// TwinCAT 3 PLC project EncapsulationPractice
// ProgramVersion: 3.1.4024.0
// libraries:
//   Tc2_Standard, * (Beckhoff Automation GmbH)
//   Tc2_System, * (Beckhoff Automation GmbH)
//   Tc3_Module, * (Beckhoff Automation GmbH)
// project tree:
//   / PlcTask.TcTTO
//   POUs/ Condition.TcPOU, FB_Bank.TcPOU, FB_IciciBank.TcPOU, MAIN.TcPOU
// (motion and I/O tree: see PLC project functionblockpractice)
// real-time tasks:
//   TASK PlcTask: cycle T#10ms, priority 20, ADS port 350
//   TASK PlcTask2: cycle T#10ms, priority 22, ADS port 352
//   TASK PlcTask1: cycle T#10ms, priority 21, ADS port 351
//   TASK PlcTask3: cycle T#10ms, priority 23, ADS port 353
//   TASK PlcTask4: cycle T#10ms, priority 24, ADS port 354
//   TASK PlcTask5: cycle T#10ms, priority 25, ADS port 355
//   TASK PlcTask6: cycle T#10ms, priority 26, ADS port 356

CONFIGURATION EncapsulationPractice
    RESOURCE PLC ON TwinCAT3
        TASK PlcTask(INTERVAL := T#10ms, PRIORITY := 25);
        PROGRAM MAIN WITH PlcTask : MAIN;
        PROGRAM Condition WITH PlcTask : Condition;
    END_RESOURCE
END_CONFIGURATION

// ---- POUs/MAIN.TcPOU
PROGRAM MAIN
VAR
	fAmount1 : REAL;
	fAmount2 : REAL;
	fbBank : FB_Bank;
	fbIciciBank : FB_IciciBank;
END_VAR

fAmount1 := fbBank.fMoney;
fbBank.sBankName := 'sbi';
fbBank.M_Deposit(4000);
fbBank.M_Withdrawal(2000);

fAmount2 := fbIciciBank.fMoney;
fbIciciBank.sBankName := 'icici';
fbIciciBank.M_Deposit(4000);
fbIciciBank.M_Withdrawal(2000);

END_PROGRAM

// ---- POUs/FB_Bank.TcPOU
FUNCTION_BLOCK FB_Bank
VAR_INPUT
	sBankName : STRING(200);
END_VAR

VAR
	fBalance : REAL;
END_VAR

{attribute 'monitoring' := 'call'}
PROPERTY fMoney : REAL
GET
fMoney := fBalance;
END_GET
SET // PRIVATE
fBalance := fMoney;
END_SET
END_PROPERTY

METHOD M_Deposit : BOOL
VAR_INPUT
	fDepositAmount : REAL;
END_VAR
fMoney := fDepositAmount;
END_METHOD

METHOD M_Withdrawal : BOOL
VAR_INPUT
	fWithdrawAmount : REAL;
END_VAR
IF fWithdrawAmount <= fMoney THEN
	fMoney := fMoney - fWithdrawAmount;
END_IF
END_METHOD

END_FUNCTION_BLOCK

// ---- POUs/FB_IciciBank.TcPOU
FUNCTION_BLOCK FB_IciciBank EXTENDS FB_Bank

VAR
END_VAR

METHOD FINAL M_Deposit : BOOL
VAR_INPUT
	fDepositAmount : REAL;
END_VAR
END_METHOD

END_FUNCTION_BLOCK

// ---- POUs/Condition.TcPOU
PROGRAM Condition
VAR
	nMark : INT := 88;
	sGrade : STRING ;
END_VAR

ACT_Case();

ACTION ACT_Case:
CASE nMark OF
	 91..100:
	sGrade := 'A';
	81..90 :
	sGrade:= 'B';
	71..80:
	sGrade:= 'C';
	61..70:
	sGrade:= 'D';
	ELSE
		sGrade:= 'F';
	
END_CASE
END_ACTION

ACTION ACT_Condition:
IF nMark > 90 THEN
	sGrade := 'A';
	ELSIF nMark > 80 THEN
		IF nMark > 85 THEN
			sGrade := 'B+';
		ELSE
			sGrade := 'B';
		END_IF
	ELSIF nMark > 70 THEN
		sGrade := 'C';
	ELSIF nMark > 60 THEN
		sGrade := 'D';
	ELSE sGrade := 'F';
END_IF
END_ACTION

END_PROGRAM
